FUNCTION_BLOCK WagoOutputBlock (* Basic Function Block Type *)
  (* Standard: 61499-2 *)
  (* Version 0.0, 2009-11-20, JHC, University of Auckland *)
  (* Compiler header: package fb.rt.wago; #include "kbusapi.h" *)
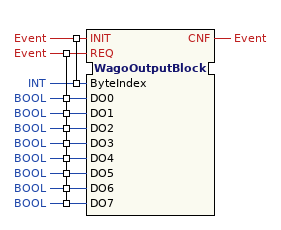
  EVENT_INPUT
    INIT WITH ByteIndex; (* Initialization Request *)
    REQ WITH DO0, DO1, DO2, DO3, DO4, DO5, DO6, DO7; (* Execution Confirmation *)
  END_EVENT
  EVENT_OUTPUT
    CNF; (* Execution Confirmation *)
  END_EVENT
  VAR_INPUT
    ByteIndex : INT;
    DO0 : BOOL;
    DO1 : BOOL;
    DO2 : BOOL;
    DO3 : BOOL;
    DO4 : BOOL;
    DO5 : BOOL;
    DO6 : BOOL;
    DO7 : BOOL;
  END_VAR
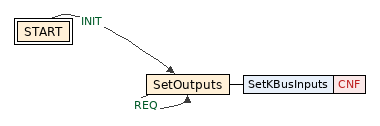
  EC_STATES
    START; (* Initial State *)
    SetOutputs : SetKBusInputs -> CNF;
  END_STATES
  EC_TRANSITIONS
    START TO SetOutputs := INIT;
    SetOutputs TO SetOutputs := REQ;
  END_TRANSITIONS
  ALGORITHM SetKBusInputs IN Java: (* Normally executed algorithm *)
// read byte from pab and show it on console
KbusOpen();

pstPabOUT->uc.Pab[me->ByteIndex] = 0x00; // CLEAR

pstPabOUT->uc.Pab[me->ByteIndex] |= me->DO0;// << 0;
pstPabOUT->uc.Pab[me->ByteIndex] |= me->DO1 << 1;
pstPabOUT->uc.Pab[me->ByteIndex] |= me->DO2 << 2;
pstPabOUT->uc.Pab[me->ByteIndex] |= me->DO3 << 3;
pstPabOUT->uc.Pab[me->ByteIndex] |= me->DO4 << 4;
pstPabOUT->uc.Pab[me->ByteIndex] |= me->DO5 << 5;
pstPabOUT->uc.Pab[me->ByteIndex] |= me->DO6 << 6;
pstPabOUT->uc.Pab[me->ByteIndex] |= me->DO7 << 7;

// Write Output values
KbusUpdate();

// Close
KbusClose();
  END_ALGORITHM
END_FUNCTION_BLOCK
